INTERFACE ITF_BaseGroupElement_HMI

END_INTERFACE

(* stored: Version 1.1.0.1
   Itf ITF_BaseGroupElement_HMI: Id {21cd6ebf-8ae8-0215-3557-71ade5490935} *)
